Omron Sysmac Studio project Odev_Video32_1 (Sysmac Studio 1.65.0.64007, StandardProject)

# Controller new_Controller_0: NX1P2-1040DT1 version 1.69
Task PrimaryTask (priority 4, period or condition 2000): Program0

VAR_GLOBAL
    BIO_Input_Bit_00 : BOOL;  (* at BuiltInIO://cpu/#0/Input_Bit_00 *)
    BIO_Input_Bit_01 : BOOL;  (* at BuiltInIO://cpu/#0/Input_Bit_01 *)
    BIO_Input_Bit_02 : BOOL;  (* at BuiltInIO://cpu/#0/Input_Bit_02 *)
    BIO_Input_Bit_03 : BOOL;  (* at BuiltInIO://cpu/#0/Input_Bit_03 *)
    BIO_Output_Bit_00 : BOOL;  (* at BuiltInIO://cpu/#0/Output_Bit_00 *)
    BIO_Output_Bit_01 : BOOL;  (* at BuiltInIO://cpu/#0/Output_Bit_01 *)
    BIO_Output_Bit_02 : BOOL;  (* at BuiltInIO://cpu/#0/Output_Bit_02 *)
    BIO_Output_Bit_03 : BOOL;  (* at BuiltInIO://cpu/#0/Output_Bit_03 *)
    IN_Start_Button : BOOL;
    IN_Stop_Button : BOOL;
    IN_OptikSensor : BOOL;
    OUT_KonveyorMotor : BOOL;
    OUT_Motor1_Start : BOOL;
    OUT_Motor2_Start : BOOL;
    Startt : BOOL;
    ServisButonu_Invert : BOOL;
    Yesil_Lamba : BOOL;
    Sari_Lamba : BOOL;
    Kirmizi_Lamba : BOOL;
    TON1_ET : TIME;
    TON2_ET : TIME;
    TON3_ET : TIME;
    StopButonu : BOOL;
    TON4_ET : TIME;
    TON5_ET : TIME;
    SecimButonu : BOOL;
END_VAR

PROGRAM Program0
VAR
    TON1 : TON;
    TON2 : TON;
    TON3 : TON;
    TON4 : TON;
    TON5 : TON;
    ı : BOOL;
END_VAR
VAR_EXTERNAL
    BIO_Input_Bit_00 : BOOL;
    BIO_Input_Bit_01 : BOOL;
    BIO_Input_Bit_02 : BOOL;
    IN_Start_Button : BOOL;
    IN_Stop_Button : BOOL;
    IN_OptikSensor : BOOL;
    OUT_KonveyorMotor : BOOL;
    BIO_Output_Bit_00 : BOOL;
    OUT_Motor1_Start : BOOL;
    BIO_Output_Bit_01 : BOOL;
    OUT_Motor2_Start : BOOL;
    BIO_Output_Bit_02 : BOOL;
    Startt : BOOL;
    ServisButonu_Invert : BOOL;
    Yesil_Lamba : BOOL;
    Sari_Lamba : BOOL;
    Kirmizi_Lamba : BOOL;
    BIO_Output_Bit_03 : BOOL;
    TON1_ET : TIME;
    TON2_ET : TIME;
    TON3_ET : TIME;
    BIO_Input_Bit_03 : BOOL;
    StopButonu : BOOL;
    TON4_ET : TIME;
    TON5_ET : TIME;
    SecimButonu : BOOL;
END_VAR

(* Section InOut: ladder, written here as Structured Text *)

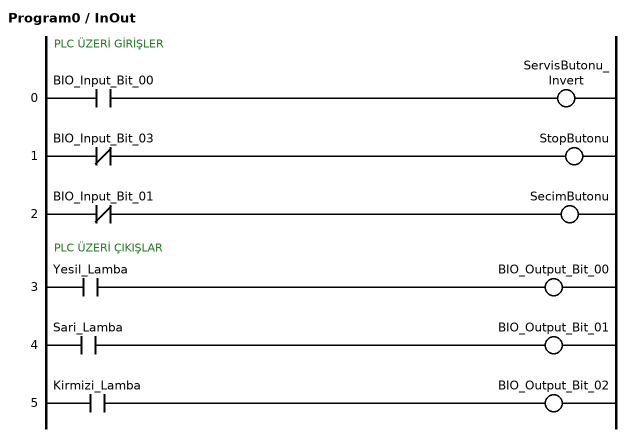
(* Rung 0: PLC ÜZERİ GİRİŞLER *)
ServisButonu_Invert := BIO_Input_Bit_00;
(* Rung 1 *)
StopButonu := NOT BIO_Input_Bit_03;
(* Rung 2 *)
SecimButonu := NOT BIO_Input_Bit_01;
(* Rung 3: PLC ÜZERİ ÇIKIŞLAR *)
BIO_Output_Bit_00 := Yesil_Lamba;
(* Rung 4 *)
BIO_Output_Bit_01 := Sari_Lamba;
(* Rung 5 *)
BIO_Output_Bit_02 := Kirmizi_Lamba;

(* Section TON_Odevi: ladder, written here as Structured Text *)

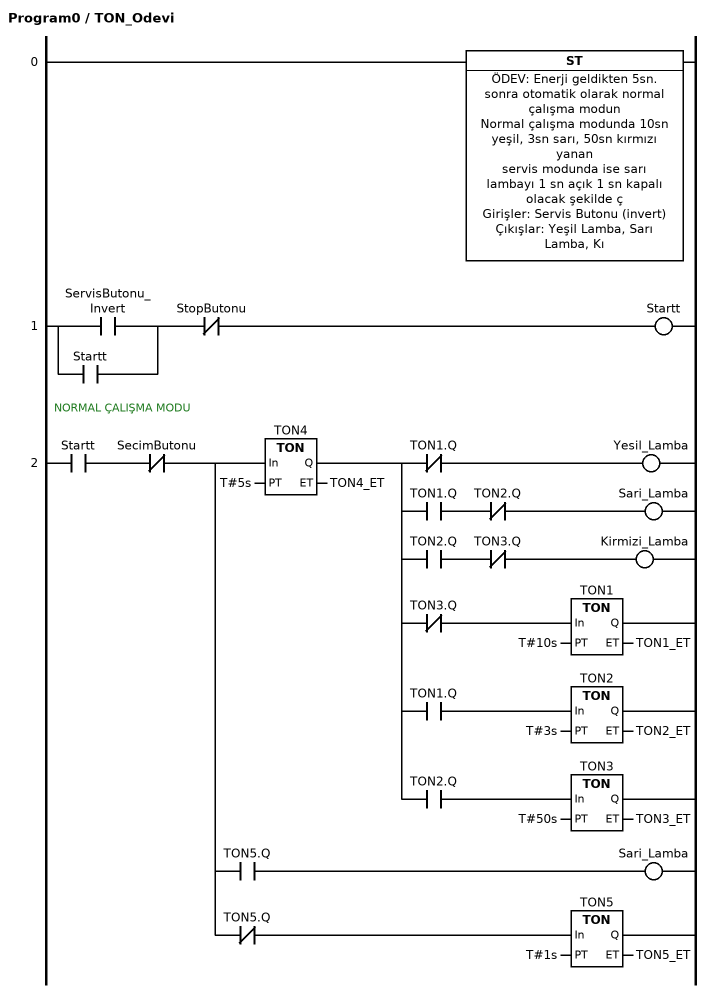
(* Rung 0 *)
ÖDEV: Enerji geldikten 5sn. sonra otomatik olarak normal çalışma moduna geçen. 
Normal çalışma modunda 10sn yeşil, 3sn sarı, 50sn kırmızı yanan 
servis modunda ise sarı lambayı 1 sn açık 1 sn kapalı olacak şekilde çalıştıran Trafik lambası PLC Programını yazınız. 
Girişler: Servis Butonu (invert) Çıkışlar: Yeşil Lamba, Sarı Lamba, Kırmızı Lamba
(* Rung 1 *)
Startt := (ServisButonu_Invert OR Startt) AND NOT StopButonu;
(* Rung 2: NORMAL ÇALIŞMA MODU *)
TON4(In := Startt AND NOT SecimButonu, PT := T#5s, ET => TON4_ET);
Yesil_Lamba := TON4.Q AND NOT TON1.Q;
Sari_Lamba := TON4.Q AND TON1.Q AND NOT TON2.Q;
Kirmizi_Lamba := TON4.Q AND TON2.Q AND NOT TON3.Q;
TON1(In := TON4.Q AND NOT TON3.Q, PT := T#10s, ET => TON1_ET);
TON2(In := TON4.Q AND TON1.Q, PT := T#3s, ET => TON2_ET);
TON3(In := TON4.Q AND TON2.Q, PT := T#50s, ET => TON3_ET);
Sari_Lamba := Startt AND NOT SecimButonu AND TON5.Q;
TON5(In := Startt AND NOT SecimButonu AND NOT TON5.Q, PT := T#1s, ET => TON5_ET);
END_PROGRAM